FUNCTION_BLOCK FB_Test
VAR_INPUT
END_VAR
VAR_OUTPUT
END_VAR
VAR
	bbb : INT;
	fb2 : FB_Test2;
END_VAR

IF Prop THEN
	bbb := 999;
END_IF

PROPERTY Prop : BOOL
GET
END_GET
SET
END_SET
END_PROPERTY

PROPERTY Prop_Out : INT
GET
Prop_Out := fb2.bOut;
END_GET
END_PROPERTY

END_FUNCTION_BLOCK

(* stored: Version 1.1.0.1, ProductVersion 3.1.4024.12
   POU FB_Test: Id {9c9b3ab2-4406-4555-87a5-09eed6bfd2c3}, SpecialFunc None
   Property Prop: Id {d1db1b66-84b6-4812-a330-f00bc0668ea9}
   Get Get: Id {39d37b2e-3072-49a8-86c4-3d7566350fbc}
   Set Set: Id {bc488e0e-37cf-44e2-972d-4cf154e9b8f1}
   Property Prop_Out: Id {cac14378-aba0-4692-b944-2ca20b8321ad}
   Get Get: Id {c9e898ca-371a-4d3a-8b68-a54429e2a874} *)
